// TwinCAT 3 PLC project OPCUA_Client
// Title: OPC UA client
// Company: Hehamala
// Author: Henri Hämäläinen
// ProjectVersion: 0.1
// Description: Tools for utitilizing PLCopen OPCUA functionalities more conveniently
// ProgramVersion: 3.1.4023.0
// libraries:
//   Tc2_Standard, * (Beckhoff Automation GmbH)
//   Tc2_System, * (Beckhoff Automation GmbH)
//   Tc3_Module, * (Beckhoff Automation GmbH)
//   Tc3_PLCopen_OpcUa, * (Beckhoff Automation GmbH)
//   TcUnit, * (www.tcunit.org)
// project tree:
//   / PlcTask.TcTTO
//   POUs/FBs/ FB_OPCUA_ClientConnection.TcPOU, FB_OPCUA_WorkOnNode.TcPOU
//   POUs/FBs/Wrappers/ UA_ConnectWrapper.TcPOU, UA_DisconnectWrapper.TcPOU, UA_GetNameSpaceIndexWrapper.TcPOU, UA_NodeGetHandleWrapper.TcPOU, UA_NodeReleaseHandleWrapper.TcPOU, UA_ReadWrapper.TcPOU, UA_WriteWrapper.TcPOU
//   POUs/ITFs/ I_OPCUA_ClientConnection.TcIO, I_OPCUA_Connect.TcIO, I_OPCUA_Disconnect.TcIO, I_OPCUA_GetNameSpaceIndex.TcIO, I_OPCUA_NodeGetHandle.TcIO, I_OPCUA_NodeReleaseHandle.TcIO, I_OPCUA_Read.TcIO, I_OPCUA_WorkOnNode.TcIO, I_OPCUA_Write.TcIO
//   POUs/Unit tests/ FB_OPCUA_ClientConnection_Test.TcPOU, FB_OPCUA_WorkOnNode_Test.TcPOU, TEST_MAIN.TcPOU
//   POUs/Unit tests/Mocks/ FB_UAconnectMock_Failure.TcPOU, FB_UAconnectMock_Success.TcPOU, FB_UAdisconnectMock_success.TcPOU, FB_UAgetNameSpaceIndexMock_success.TcPOU, FB_UAnodeGetHandleMock_Success.TcPOU, FB_UAnodeReleaseHandleMock_Success.TcPOU, FB_UAreadMock_BoolChangesToTrue.TcPOU, FB_UAwriteMock_Failure.TcPOU
//   Version/ Global_Version.TcGVL
// real-time tasks:
//   TASK PlcTask: cycle T#10ms, priority 20, ADS port 350

CONFIGURATION OPCUA_Client
    RESOURCE PLC ON TwinCAT3
        TASK PlcTask(INTERVAL := T#10ms, PRIORITY := 20);
        PROGRAM TEST_MAIN WITH PlcTask : TEST_MAIN;
    END_RESOURCE
END_CONFIGURATION

// ---- Version/Global_Version.TcGVL
{attribute 'TcGenerated'}
{attribute 'no-analysis'}
{attribute 'linkalways'}
// This function has been automatically generated from the project information.
VAR_GLOBAL CONSTANT
	{attribute 'const_non_replaced'}
	stLibVersion_OPC_UA_client : ST_LibVersion := (iMajor := 0, iMinor := 1, iBuild := 0, iRevision := 0, nFlags := 0, sVersion := '0.1');
END_VAR

// ---- POUs/ITFs/I_OPCUA_ClientConnection.TcIO
INTERFACE I_OPCUA_ClientConnection

METHOD connect : BOOL
VAR_INPUT
	(* server address *)
	serverUrl 		: STRING(MAX_STRING_LENGTH); 
	(* namespace uri*)
	namespaceUri	: STRING(MAX_STRING_LENGTH);
	(* Location of data in namespace *)
	nameSpaceLocationIdentifier : STRING(MAX_STRING_LENGTH);
	(* Session connect info struct *)
	sessionConnectInfo	: ST_UASessionConnectInfo;
END_VAR
END_METHOD

METHOD disconnect : BOOL
END_METHOD

END_INTERFACE

// ---- POUs/ITFs/I_OPCUA_Connect.TcIO
INTERFACE I_OPCUA_Connect

METHOD start : BOOL
VAR_INPUT
    Execute            : BOOL;
    ServerUrl          : STRING(MAX_STRING_LENGTH);
    SessionConnectInfo : ST_UASessionConnectInfo;     
    Timeout            : TIME := DEFAULT_ADS_TIMEOUT; 
END_VAR
VAR_OUTPUT
    ConnectionHdl : DWORD;
    Done          : BOOL;
    Busy          : BOOL;
    Error         : BOOL;
    ErrorID       : DWORD;
END_VAR
END_METHOD

END_INTERFACE

// ---- POUs/ITFs/I_OPCUA_Disconnect.TcIO
INTERFACE I_OPCUA_Disconnect

METHOD start : BOOL
VAR_INPUT
    Execute           : BOOL;
    ConnectionHdl     : DWORD;     
    Timeout           : TIME := DEFAULT_ADS_TIMEOUT; 
END_VAR 
VAR_OUTPUT
    Done        : BOOL;
    Busy        : BOOL;
    Error       : BOOL;
    ErrorID     : DWORD;
END_VAR
END_METHOD

END_INTERFACE

// ---- POUs/ITFs/I_OPCUA_GetNameSpaceIndex.TcIO
INTERFACE I_OPCUA_GetNameSpaceIndex

METHOD start : BOOL
VAR_INPUT
    Execute       : BOOL;
    ConnectionHdl : DWORD;
    NamespaceUri  : STRING(MAX_STRING_LENGTH);
    Timeout       : TIME := DEFAULT_ADS_TIMEOUT; 
END_VAR
VAR_OUTPUT
    NamespaceIndex : UINT;
    Done           : BOOL;
    Busy           : BOOL;
    Error          : BOOL;
    ErrorID        : DWORD;
END_VAR
END_METHOD

END_INTERFACE

// ---- POUs/ITFs/I_OPCUA_NodeGetHandle.TcIO
INTERFACE I_OPCUA_NodeGetHandle

METHOD start : BOOL
VAR_INPUT
    Execute       : BOOL;
    ConnectionHdl : DWORD;
    NodeID        : ST_UANodeID;
    Timeout       : TIME := DEFAULT_ADS_TIMEOUT; 
END_VAR 
VAR_OUTPUT
    NodeHdl     : DWORD;
    Done        : BOOL;
    Busy        : BOOL;
    Error       : BOOL;
    ErrorID     : DWORD;
END_VAR
END_METHOD

END_INTERFACE

// ---- POUs/ITFs/I_OPCUA_NodeReleaseHandle.TcIO
INTERFACE I_OPCUA_NodeReleaseHandle

METHOD start : BOOL
VAR_INPUT
    Execute       : BOOL;
    ConnectionHdl : DWORD;
    NodeHdl       : DWORD;
    Timeout       : TIME := DEFAULT_ADS_TIMEOUT; 
END_VAR 
VAR_OUTPUT
    Done       : BOOL;
    Busy       : BOOL;
    Error      : BOOL;
    ErrorID    : DWORD;
END_VAR
END_METHOD

END_INTERFACE

// ---- POUs/ITFs/I_OPCUA_Read.TcIO
INTERFACE I_OPCUA_Read

METHOD start : BOOL
VAR_INPUT
    Execute           : BOOL;
    ConnectionHdl     : DWORD;
    NodeHdl           : DWORD;
    stNodeAddInfo     : ST_UANodeAdditionalInfo;
    pVariable         : PVOID;
    cbData            : UDINT;
    Timeout           : TIME := DEFAULT_ADS_TIMEOUT;    
END_VAR 
VAR_OUTPUT
    Done        : BOOL;
    Busy        : BOOL;
    Error       : BOOL;
    ErrorID     : UDINT;
    cbData_R    : UDINT;
END_VAR
END_METHOD

END_INTERFACE

// ---- POUs/ITFs/I_OPCUA_WorkOnNode.TcIO
INTERFACE I_OPCUA_WorkOnNode

METHOD read : BOOL
VAR_INPUT
	//clientVariable	: ANY;
	(* VAR_INFO of the target variable (from GVL_OPC)*)
	//clientVariableInfo	: __SYSTEM.VAR_INFO;
	clientVariableAddress	: PVOID;
	clientVariableSize : UDINT;
	serverNodeIdentifier	: STRING;
	nameSpaceLocationIdentifierEx : STRING(MAX_STRING_LENGTH);
	connectionHdl : DWORD;
	nNamespaceIndex			: UINT;
END_VAR
END_METHOD

METHOD write : BOOL
VAR_INPUT
	//clientVariable	: ANY;
	(* VAR_INFO of the target variable (from GVL_OPC)*)
	//clientVariableInfo	: __SYSTEM.VAR_INFO;
	clientVariableAddress	: PVOID;
	clientVariableSize : UDINT;
	serverNodeIdentifier	: STRING;
	nameSpaceLocationIdentifierEx : STRING(MAX_STRING_LENGTH);
	connectionHdl : DWORD;
	nNamespaceIndex			: UINT;
END_VAR
END_METHOD

END_INTERFACE

// ---- POUs/ITFs/I_OPCUA_Write.TcIO
INTERFACE I_OPCUA_Write

METHOD start : BOOL
VAR_INPUT
    Execute        : BOOL;
    ConnectionHdl  : DWORD;
    NodeHdl        : DWORD;
    stNodeAddInfo  : ST_UANodeAdditionalInfo; 
    pVariable      : PVOID;
    cbData         : UDINT;     
    Timeout        : TIME := DEFAULT_ADS_TIMEOUT; 
END_VAR 
VAR_OUTPUT
    Done      : BOOL;
    Busy      : BOOL;
    Error     : BOOL;
    ErrorID   : DWORD;
END_VAR
END_METHOD

END_INTERFACE

// ---- POUs/Unit tests/TEST_MAIN.TcPOU
PROGRAM TEST_MAIN
VAR
	clientConnectionTest 	: FB_OPCUA_ClientConnection_Test;
	workOnNodeTest			: FB_OPCUA_WorkOnNode_Test;
	startTest				: BOOL;
END_VAR


IF startTest THEN
	TcUnit.RUN();
END_IF

END_PROGRAM

// ---- POUs/Unit tests/FB_OPCUA_ClientConnection_Test.TcPOU
FUNCTION_BLOCK FB_OPCUA_ClientConnection_Test  EXTENDS TcUnit.FB_TestSuite
VAR_INPUT
END_VAR
VAR_OUTPUT
END_VAR
VAR
END_VAR

errorShouldntBeActiveWhenConnectionIsSuccesful();
errorShouldBeActiveIfConnectingFails();

METHOD errorShouldBeActiveIfConnectingFails
VAR
	connect 				: FB_UAconnectMock_Failure;
	disconnect 				: FB_UAdisconnectMock_success;
	getNameSpaceIndex 		: FB_UAgetNameSpaceIndexMock_success;
	connection 				: FB_OPCUA_ClientConnection(iOPCUAconnect := connect,
														iOPCUAdisconnect := disconnect,
														iOPCUAgetNameSpaceIndex := getNameSpaceIndex);
	sessionCOnnectInfo 		: ST_UASessionConnectInfo;
END_VAR
TEST('errorShouldBeActiveIfConnectingFails');
	connection.connect(serverUrl := '11.11.11.11',
				namespaceUri := 'namespace',
				nameSpaceLocationIdentifier := 'GVL_ident' ,
				sessionConnectInfo := SessionConnectInfo
				);
	assertEquals_BOOL(Expected := TRUE, Actual := connection.error, Message := 'Error not active when connection failed');
TEST_FINISHED();
END_METHOD

METHOD errorShouldntBeActiveWhenConnectionIsSuccesful
VAR
	connect : FB_UAconnectMock_Success;
	disconnect : FB_UAdisconnectMock_success;
	getNameSpaceIndex : FB_UAgetNameSpaceIndexMock_success;
	connection : FB_OPCUA_ClientConnection(iOPCUAconnect := connect,
										iOPCUAdisconnect := disconnect,
										iOPCUAgetNameSpaceIndex := getNameSpaceIndex);
	sessionCOnnectInfo : ST_UASessionConnectInfo;
END_VAR
TEST('errorShouldntBeActiveWhenConnectionIsSuccesful');
	connection.connect(serverUrl := '11.11.11.11',
				namespaceUri := 'namespace',
				nameSpaceLocationIdentifier := 'GVL_ident' ,
				sessionConnectInfo := SessionConnectInfo
				);
	assertEquals_BOOL(Expected := FALSE, Actual := connection.error, Message := 'Error active even when connection succeeced');
TEST_FINISHED();
END_METHOD

END_FUNCTION_BLOCK

// ---- POUs/Unit tests/Mocks/FB_UAconnectMock_Failure.TcPOU
FUNCTION_BLOCK FB_UAconnectMock_Failure IMPLEMENTS I_OPCUA_Connect
VAR_INPUT
END_VAR
VAR_OUTPUT
END_VAR
VAR
END_VAR

{warning 'add method implementation '}
METHOD start : BOOL
VAR_INPUT
	Execute	: BOOL;
	ServerUrl	: STRING(MAX_STRING_LENGTH);
	SessionConnectInfo	: Tc3_PLCopen_OpcUa.ST_UASessionConnectInfo;
	Timeout	: TIME := DEFAULT_ADS_TIMEOUT;
END_VAR
VAR_OUTPUT
	ConnectionHdl	: DWORD;
	Done	: BOOL;
	Busy	: BOOL;
	Error	: BOOL;
	ErrorID	: DWORD;
END_VAR
IF execute THEN
	error := TRUE;
END_IF
END_METHOD

END_FUNCTION_BLOCK

// ---- POUs/Unit tests/Mocks/FB_UAdisconnectMock_success.TcPOU
FUNCTION_BLOCK FB_UAdisconnectMock_success IMPLEMENTS I_OPCUA_Disconnect
VAR_INPUT
END_VAR
VAR_OUTPUT
END_VAR
VAR
END_VAR

{warning 'add method implementation '}
METHOD start : BOOL
VAR_INPUT
	Execute	: BOOL;
	ConnectionHdl	: DWORD;
	Timeout	: TIME := DEFAULT_ADS_TIMEOUT;
END_VAR
VAR_OUTPUT
	Done	: BOOL;
	Busy	: BOOL;
	Error	: BOOL;
	ErrorID	: DWORD;
END_VAR
IF execute THEN
	done := TRUE;
END_IF
END_METHOD

END_FUNCTION_BLOCK

// ---- POUs/Unit tests/Mocks/FB_UAgetNameSpaceIndexMock_success.TcPOU
FUNCTION_BLOCK FB_UAgetNameSpaceIndexMock_success IMPLEMENTS I_OPCUA_GetNameSpaceIndex
VAR_INPUT
END_VAR
VAR_OUTPUT
END_VAR
VAR
END_VAR

{warning 'add method implementation '}
METHOD start : BOOL
VAR_INPUT
	Execute	: BOOL;
	ConnectionHdl	: DWORD;
	NamespaceUri	: STRING(MAX_STRING_LENGTH);
	Timeout	: TIME := DEFAULT_ADS_TIMEOUT;
END_VAR
VAR_OUTPUT
	NamespaceIndex	: UINT;
	Done	: BOOL;
	Busy	: BOOL;
	Error	: BOOL;
	ErrorID	: DWORD;
END_VAR
IF execute THEN
	done := TRUE;
END_IF
END_METHOD

END_FUNCTION_BLOCK

// ---- POUs/FBs/FB_OPCUA_ClientConnection.TcPOU
FUNCTION_BLOCK FB_OPCUA_ClientConnection IMPLEMENTS I_OPCUA_ClientConnection
VAR_INPUT
END_VAR
VAR_OUTPUT
	connectionHdl : DWORD;
	nNamespaceIndex			: UINT;
	connectDone : BOOL;
	disconnectDone : BOOL;
	error : BOOL;
END_VAR
VAR
	nameSpaceLocationIdentifierEx : STRING(MAX_STRING_LENGTH); 
	NamespaceUriEx : STRING(MAX_STRING_LENGTH); 
	
	{IF defined (Test)}	
		_iOPCUA_Connect				: I_OPCUA_COnnect;
		_iOPCUA_GetNameSpaceIndex 	: I_OPCUA_GetNameSpaceIndex;
		_iOPCUA_Disconnect			: I_OPCUA_Disconnect;
	{ELSE}
		_iOPCUA_Connect				: UA_ConnectWrapper;		
		_iOPCUA_GetNameSpaceIndex 	: UA_GetNameSpaceIndexWrapper;
		_iOPCUA_Disconnect			: UA_DisconnectWrapper;
	{END_IF}
		
	SessionConnectInfoEx	: ST_UASessionConnectInfo;
	
	

	
	(* Other declarations *) 
	errorID : DWORD;	
	executing : BOOL;
	firstTimeWrite : BOOL;
	serverURLex: STRING(MAX_STRING_LENGTH);
	connectStep: INT;
	disconnectStep: INT;
	connectBusy: BOOL;
	connectError: BOOL;
	getNameSpaceIndexBusy: BOOL;
	getNameSpaceIndexError: BOOL;
	disconnectBusy: BOOL;
	disconnectError: BOOL;
	getNameSpaceErrorID: DWORD;
	connectErrorID: DWORD;
END_VAR

{warning 'add method implementation '}
METHOD connect : BOOL
VAR_INPUT
	(* server address *)
	serverUrl	: STRING(MAX_STRING_LENGTH);
	(* namespace uri*)
	namespaceUri	: STRING(MAX_STRING_LENGTH);
	(* Location of data in namespace *)
	nameSpaceLocationIdentifier	: STRING(MAX_STRING_LENGTH);
	(* Session connect info struct *)
	sessionConnectInfo	: ST_UASessionConnectInfo;
END_VAR


CASE connectStep OF
	0:
		error := FALSE;
		connectDone := FALSE;
		disconnectStep := 0;
		nameSpaceUriEx := namespaceUri;
		sessionConnectInfoEx := SessionConnectInfo;
		serverURlex := serverUrl;
		nameSpaceLocationIdentifierEx := nameSpaceLocationIdentifier;
		SessionConnectInfoEx.sApplicationName := 'asddddd';
		_iOPCUA_Connect.start(
			Execute				:= TRUE,
			ServerURL			:= serverURLex,
			SessionConnectInfo  := SessionConnectInfoEx,
			Timeout				:= T#2M,
			ConnectionHdl		=> ConnectionHdl,
			busy				=> connectBusy,
			error				=> connectError,
			errorID				=> connectErrorID
		);
		IF NOT connectBusy THEN
			_iOPCUA_Connect.start(Execute := FALSE,
								ServerURL			:= serverURLex,
								SessionConnectInfo  := SessionConnectInfoEx,
								Timeout				:= T#2M,
								ConnectionHdl		=> ConnectionHdl
								);
	
			IF NOT connectError THEN
				(* session open *)
				connectStep :=connectStep + 1;
			ELSE
				Error			:= TRUE;
				ErrorID		:= connectErrorID;
				ConnectionHdl	:= 0;
				connectStep		:= 0; (* idle *)
			END_IF
		END_IF
	1:
		_iOPCUA_GetNameSpaceIndex.start(
										Execute			:= TRUE,
										ConnectionHdl	:= ConnectionHdl,
										NamespaceUri	:= NamespaceUriEx,
										TimeOut 		:= T#5S,
										NamespaceIndex	=> nNamespaceIndex,
										busy			=> getNameSpaceIndexBusy,
										error			=> getNameSpaceIndexError,
										errorID			=> getNameSpaceErrorID
										);
	
	
		IF NOT getNameSpaceIndexBusy THEN
			_iOPCUA_GetNameSpaceIndex.start(Execute := FALSE,
											ConnectionHdl	:= ConnectionHdl,
											NamespaceUri	:= NamespaceUriEx,
											TimeOut 		:= T#5S,
											NamespaceIndex	=> nNamespaceIndex,
											);
			IF NOT getNameSpaceIndexError THEN
				(* session closed *)
				connectDone := TRUE;
				connectStep 	:= 0; (* idle *)
			ELSE
				Error		:= TRUE;
				ErrorID	:= getNameSpaceErrorID;
				connectStep := 0;
				// CLEANUP?writeStep 		:= 5; (* idle *)
			END_IF
		END_IF	
END_CASE
END_METHOD

{warning 'add method implementation '}
METHOD disconnect : BOOL

VAR
	Execute: INT;
	disconnectErrorID: DWORD;
END_VAR
CASE disconnectStep OF
	0:	(* close session *)
		error := FALSE;
		disconnectDone := FALSE;
		connectStep := 0;
		_iOPCUA_Disconnect.start(
							Execute			:= TRUE,
							ConnectionHdl	:= connectionHdl,
							timeOut			:= T#5S,
							busy			=> disconnectBusy,
							error			=> disconnectError,
							errorID			=> disconnectErrorID
						);
	
		IF NOT disconnectBusy THEN
			_iOPCUA_Disconnect.start(Execute := FALSE,
									ConnectionHdl	:= connectionHdl,
									timeOut			:= T#5S
									);
			//Busy := FALSE;
			IF NOT disconnectError THEN
				(* session closed *)
				firstTimeWrite := TRUE;
				Executing := FALSE;
				ConnectionHdl	:= 0; //ADDED
				disconnectStep 		:= 0; (* idle *)
				IF NOT error THEN 
					disconnectDone := TRUE;
					disconnectStep := 0;
				END_IF
			ELSE
				error			:= TRUE;
				errorID		:= disconnectErrorID;
				connectionHdl	:= 0;
				disconnectStep 		:= 0; 
			END_IF
		END_IF	
END_CASE
END_METHOD

METHOD FB_init : BOOL
VAR_INPUT
	bInitRetains					: BOOL; // if TRUE, the retain variables are initialized (warm start / cold start)
	bInCopyCode 					: BOOL;  // if TRUE, the instance afterwards gets moved into the copy code (online change)
	{IF defined (Test)}
		iOPCUAconnect 					: I_OPCUA_Connect;
		iOPCUAdisconnect 				: I_OPCUA_Disconnect;
		iOPCUAgetNameSpaceIndex 		: I_OPCUA_GetNameSpaceIndex; 
	{ END_IF }
END_VAR
{IF defined (Test)}
	_iOPCUA_Connect := iOPCUAconnect;
	_iOPCUA_Disconnect := iOPCUAdisconnect;
	_iOPCUA_GetNameSpaceIndex := iOPCUAgetNameSpaceIndex;
{ END_IF }
END_METHOD

END_FUNCTION_BLOCK

// ---- POUs/FBs/Wrappers/UA_ConnectWrapper.TcPOU
FUNCTION_BLOCK UA_ConnectWrapper IMPLEMENTS I_OPCUA_Connect
VAR_INPUT
END_VAR
VAR_OUTPUT
END_VAR
VAR
	uaConnect : UA_Connect;
END_VAR

{warning 'add method implementation '}
METHOD start : BOOL
VAR_INPUT
	Execute					: BOOL;
	ServerUrl				: STRING(MAX_STRING_LENGTH);
	SessionConnectInfo		: Tc3_PLCopen_OpcUa.ST_UASessionConnectInfo;
	Timeout					: TIME := DEFAULT_ADS_TIMEOUT;
END_VAR
VAR_OUTPUT
	ConnectionHdl			: DWORD;
	Done					: BOOL;
	Busy					: BOOL;
	Error					: BOOL;
	ErrorID					: DWORD;
END_VAR
uaConnect(Execute					:= Execute,
          ServerUrl				:= ServerUrl	,
          SessionConnectInfo		:= SessionConnectInfo,
          Timeout					:= Timeout,
		  ConnectionHdl			=> ConnectionHdl,
		  Done					=> Done,
          Busy					=> Busy,
          Error					=> Error,
          ErrorID				=> ErrorID
		  );
END_METHOD

END_FUNCTION_BLOCK

// ---- POUs/FBs/Wrappers/UA_GetNameSpaceIndexWrapper.TcPOU
FUNCTION_BLOCK UA_GetNameSpaceIndexWrapper IMPLEMENTS I_OPCUA_GetNameSpaceIndex
VAR_INPUT
END_VAR
VAR_OUTPUT
END_VAR
VAR
	uaGetNameSpaceIndex : UA_GetNameSpaceIndex;
END_VAR

{warning 'add method implementation '}
METHOD start : BOOL
VAR_INPUT
	Execute			: BOOL;
	ConnectionHdl	: DWORD;
	NamespaceUri	: STRING(MAX_STRING_LENGTH);
	Timeout			: TIME := DEFAULT_ADS_TIMEOUT;
END_VAR
VAR_OUTPUT
	NamespaceIndex	: UINT;
	Done			: BOOL;
	Busy			: BOOL;
	Error			: BOOL;
	ErrorID			: DWORD;
END_VAR
uaGetNameSpaceIndex(Execute			:= Execute,
                    ConnectionHdl	:= ConnectionHdl,
                    NamespaceUri	:= Namespaceuri,
                    Timeout			:= Timeout,
					NamespaceIndex	=> NamespaceIndex,
                    Done			=> Done,
                    Busy			=> Busy,
                    Error			=> Error,
                    ErrorID			=> ErrorID);
END_METHOD

END_FUNCTION_BLOCK

// ---- POUs/FBs/Wrappers/UA_DisconnectWrapper.TcPOU
FUNCTION_BLOCK UA_DisconnectWrapper IMPLEMENTS I_OPCUA_Disconnect
VAR_INPUT
END_VAR
VAR_OUTPUT
END_VAR
VAR
	uaDisconnect : UA_Disconnect;
END_VAR

{warning 'add method implementation '}
METHOD start : BOOL
VAR_INPUT
	Execute			: BOOL;
	ConnectionHdl	: DWORD;
	Timeout			: TIME := DEFAULT_ADS_TIMEOUT;
END_VAR
VAR_OUTPUT
	Done	: BOOL;
	Busy	: BOOL;
	Error	: BOOL;
	ErrorID	: DWORD;
END_VAR
uaDisconnect(Execute			:= Execute,
             ConnectionHdl	:= ConnectionHdl,
             Timeout			:= Timeout,
			 Done			=> Done,
			 Busy			=> Busy,
             Error			=> Error,
             ErrorID 		=> ErrorID);
END_METHOD

END_FUNCTION_BLOCK

// ---- POUs/Unit tests/Mocks/FB_UAconnectMock_Success.TcPOU
FUNCTION_BLOCK FB_UAconnectMock_Success IMPLEMENTS I_OPCUA_Connect
VAR_INPUT
END_VAR
VAR_OUTPUT
END_VAR
VAR
END_VAR

{warning 'add method implementation '}
METHOD start : BOOL
VAR_INPUT
	Execute	: BOOL;
	ServerUrl	: STRING(MAX_STRING_LENGTH);
	SessionConnectInfo	: Tc3_PLCopen_OpcUa.ST_UASessionConnectInfo;
	Timeout	: TIME := DEFAULT_ADS_TIMEOUT;
END_VAR
VAR_OUTPUT
	ConnectionHdl	: DWORD;
	Done	: BOOL;
	Busy	: BOOL;
	Error	: BOOL;
	ErrorID	: DWORD;
END_VAR
IF execute THEN
	done := TRUE;
END_IF
END_METHOD

END_FUNCTION_BLOCK

// ---- POUs/Unit tests/FB_OPCUA_WorkOnNode_Test.TcPOU
FUNCTION_BLOCK FB_OPCUA_WorkOnNode_Test  EXTENDS TcUnit.FB_TestSuite
VAR_INPUT
END_VAR
VAR_OUTPUT
END_VAR
VAR
	read	 				: FB_UAreadMock_BoolChangesToTrue;
	write					: FB_UAwriteMock_Failure;
	nodeReleaseHandle		: FB_UAnodeReleaseHandleMock_Success;
	nodeGetHandle			: FB_UAnodeGetHandleMock_Success;

	readNode 				: FB_OPCUA_WorkOnNode(
													iOPCUA_Write := write,			
													iOPCUA_Read	:= read,				
													iOPCUA_NodeReleaseHandle := nodeReleaseHandle,	
													iOPCUA_NodeGetHandle :=  nodeGetHandle		
													);
	booleanToRead : BOOL;
	booleanInfo : __SYSTEM.VAR_INFO := __VARINFO(readNode);
END_VAR

variableShouldGetUpdatedWhenChanged();

METHOD errorShouldActivateIfWriteFails
VAR
	sessionCOnnectInfo 		: ST_UASessionConnectInfo;
END_VAR
END_METHOD

METHOD variableShouldGetUpdatedWhenChanged
VAR
	sessionCOnnectInfo 		: ST_UASessionConnectInfo;
END_VAR
TEST('variableShouldGetUpdatedWhenChanged');
	
	
	readNode.read(//clientVariable := booleanToRead,
					clientVariableAddress := ADR(booleanToRead),
					clientVariableSize := SIZEOF(booleanToRead),
					serverNodeIdentifier := 'test',
					nameSpaceLocationIdentifierEx := 'test',
					ConnectionHdl := 11,
					nNamespaceIndex := 11);
	IF NOT readNode.busy THEN
		assertEquals_BOOL(Expected := TRUE, Actual := booleanToRead, Message := 'Value not updated when changed');
		TEST_FINISHED();
	END_IF
END_METHOD

END_FUNCTION_BLOCK

// ---- POUs/Unit tests/Mocks/FB_UAreadMock_BoolChangesToTrue.TcPOU
FUNCTION_BLOCK FB_UAreadMock_BoolChangesToTrue IMPLEMENTS I_OPCUA_Read
VAR_INPUT
END_VAR
VAR_OUTPUT
END_VAR
VAR
END_VAR

{warning 'add method implementation '}
METHOD start : BOOL
VAR_INPUT
	Execute	: BOOL;
	ConnectionHdl	: DWORD;
	NodeHdl	: DWORD;
	stNodeAddInfo	: Tc3_PLCopen_OpcUa.ST_UANodeAdditionalInfo;
	pVariable	: PVOID;
	cbData	: UDINT;
	Timeout	: TIME := DEFAULT_ADS_TIMEOUT;
END_VAR
VAR_OUTPUT
	Done	: BOOL;
	Busy	: BOOL;
	Error	: BOOL;
	ErrorID	: UDINT;
	cbData_R	: UDINT;
END_VAR
IF execute THEN
	MEMSET(pVariable,1,SIZEOF(cbData));
	done := TRUE;
END_IF
END_METHOD

END_FUNCTION_BLOCK

// ---- POUs/Unit tests/Mocks/FB_UAwriteMock_Failure.TcPOU
FUNCTION_BLOCK FB_UAwriteMock_Failure IMPLEMENTS I_OPCUA_Write
VAR_INPUT
END_VAR
VAR_OUTPUT
END_VAR
VAR
END_VAR

{warning 'add method implementation '}
METHOD start : BOOL
VAR_INPUT
	Execute	: BOOL;
	ConnectionHdl	: DWORD;
	NodeHdl	: DWORD;
	stNodeAddInfo	: Tc3_PLCopen_OpcUa.ST_UANodeAdditionalInfo;
	pVariable	: PVOID;
	cbData	: UDINT;
	Timeout	: TIME := DEFAULT_ADS_TIMEOUT;
END_VAR
VAR_OUTPUT
	Done	: BOOL;
	Busy	: BOOL;
	Error	: BOOL;
	ErrorID	: DWORD;
END_VAR
IF execute THEN
	Error := TRUE;
END_IF
END_METHOD

END_FUNCTION_BLOCK

// ---- POUs/Unit tests/Mocks/FB_UAnodeReleaseHandleMock_Success.TcPOU
FUNCTION_BLOCK FB_UAnodeReleaseHandleMock_Success IMPLEMENTS I_OPCUA_NodeReleaseHandle
VAR_INPUT
END_VAR
VAR_OUTPUT
END_VAR
VAR
END_VAR

{warning 'add method implementation '}
METHOD start : BOOL
VAR_INPUT
    Execute       : BOOL;
    ConnectionHdl : DWORD;
    NodeHdl       : DWORD;
    Timeout       : TIME := DEFAULT_ADS_TIMEOUT; 
END_VAR
VAR_OUTPUT
	Done	: BOOL;
	Busy	: BOOL;
	Error	: BOOL;
	ErrorID	: DWORD;
END_VAR
IF execute THEN
	done := TRUE;
END_IF
END_METHOD

END_FUNCTION_BLOCK

// ---- POUs/Unit tests/Mocks/FB_UAnodeGetHandleMock_Success.TcPOU
FUNCTION_BLOCK FB_UAnodeGetHandleMock_Success IMPLEMENTS I_OPCUA_NodeGetHandle
VAR_INPUT
END_VAR
VAR_OUTPUT
END_VAR
VAR
END_VAR

{warning 'add method implementation '}
METHOD start : BOOL
VAR_INPUT
	Execute	: BOOL;
	ConnectionHdl	: DWORD;
	NodeID	: Tc3_PLCopen_OpcUa.ST_UANodeID;
	Timeout	: TIME := DEFAULT_ADS_TIMEOUT;
END_VAR
VAR_OUTPUT
	NodeHdl	: DWORD;
	Done	: BOOL;
	Busy	: BOOL;
	Error	: BOOL;
	ErrorID	: DWORD;
END_VAR
IF execute THEN
	Done := TRUE;
END_IF
END_METHOD

END_FUNCTION_BLOCK

// ---- POUs/FBs/FB_OPCUA_WorkOnNode.TcPOU
FUNCTION_BLOCK FB_OPCUA_WorkOnNode IMPLEMENTS I_OPCUA_WorkOnNode
VAR_INPUT
END_VAR
VAR_OUTPUT
	busy: BOOL;
	error : BOOL;
END_VAR
VAR

	stNodeAddInfo			: ST_UANodeAdditionalInfo;
	cbData_R				: UDINT;
	
	iState		: INT;
	nErrorID	: DWORD;
	lastErrorStep: INT;
	Executing : BOOL;
	writeStep : INT;
	(* Declarations for UA_Write *)
	{IF defined (Test)}
		_iOPCUA_Write : I_OPCUA_Write; 
		(* Declarations for UA_NodeReleaseHandle *)
		_iOPCUA_NodeReleaseHandle : I_OPCUA_NodeReleaseHandle;
		_iOPCUA_NodeGetHandle : I_OPCUA_NodeGetHandle;
		_iOPCUA_Read			: I_OPCUA_Read;
	{ELSE}
		_iOPCUA_Write : UA_WriteWrapper;
		_iOPCUA_NodeReleaseHandle : UA_NOdeReleaseHandleWrapper;
		_iOPCUA_NodeGetHandle : UA_NodeGetHandleWrapper;
		_iOPCUA_Read			: UA_ReadWrapper;
	{ END_IF}
	(* Other declarations *) 
	errorID : DWORD;	
	clientVariablePrev : BYTE;
	firstTimeWrite : BOOL;
	//_iOPCUA_NodeGetHandle : I_OPCUA_NodeGetHandle;
	NodeID : ST_UANodeID;
	nNodeHdl : DWORD;
	NodeGetHandleBusy: BOOL;
	NodeGetHandleError: BOOL;
	NodeGetHandleErrorID: DWORD;
	readBusy: BOOL;
	readError: BOOL;
	readErrorID: DWORD;
	nodeReleaseHandleBusy: BOOL;
	nodeReleaseHandleError: BOOL;
	nodeReleaseHandleErrorID: DWORD;
	writeBusy: BOOL;
	writeError: BOOL;
	writeErrorID: DWORD;
	clientVarInfo : __SYSTEM.VAR_INFO;
	pClientByteValue : POINTER TO BYTE;
	ConnectionHdlPrev: DWORD;
END_VAR

METHOD FB_init : BOOL
VAR_INPUT
	bInitRetains : BOOL; // if TRUE, the retain variables are initialized (warm start / cold start)
	bInCopyCode : BOOL;  // if TRUE, the instance afterwards gets moved into the copy code (online change)
	{IF defined (Test)}
		iOPCUA_Write				: I_OPCUA_Write;
		iOPCUA_Read					: I_OPCUA_Read;
		iOPCUA_NodeReleaseHandle 	: I_OPCUA_NodeReleaseHandle;
		iOPCUA_NodeGetHandle 		: I_OPCUA_NodeGetHandle;
	{END_IF}
END_VAR
{IF defined (Test)}
	_iOPCUA_Write	:= iOPCUA_Write;		
	_iOPCUA_Read		:= iOPCUA_Read	;		
	_iOPCUA_NodeReleaseHandle := iOPCUA_NodeReleaseHandle;
	_iOPCUA_NodeGetHandle 	:= iOPCUA_NodeGetHandle 	;
{END_IF}
END_METHOD

{warning 'add method implementation '}
METHOD read : BOOL
VAR_INPUT
	{attribute 'anytypeclass' := 'ANY'}
	//clientVariable	: ANY;
	(* VAR_INFO of the target variable (from GVL_OPC)*)
	//clientVariableInfo	: __SYSTEM.VAR_INFO;
	clientVariableAddress : PVOID;
	clientVariableSize : UDINT;
	serverNodeIdentifier	: STRING;
	nameSpaceLocationIdentifierEx	: STRING(MAX_STRING_LENGTH);
	ConnectionHdl	: DWORD;
	nNamespaceIndex			: UINT;
END_VAR

IF ConnectionHdl <> ConnectionHdlPrev THEN
	istate := 0;
	ConnectionHdlPrev := ConnectionHdl;
	error := FALSE;
END_IF

CASE istate OF
0: 
		error := FALSE;
		nNodeHdl :=0;
		iState := iState + 1;
		Executing := TRUE;
	
1:	(* Get Node Handle *)
	
		NodeID.eIdentifierType := eUAIdentifierType_String;
		NodeID.nNamespaceIndex := nNamespaceIndex;
		NodeID.sIdentifier := CONCAT(nameSpaceLocationIdentifierEx,serverNodeIdentifier);
		_iOPCUA_NodeGetHandle.start(
									Execute := TRUE,
									ConnectionHdl := connectionHdl,
									NodeID := NodeID,
									Timeout := T#5S,
									NodeHdl => nNodeHdl,
									Busy => NodeGetHandleBusy,
									Error => NodeGetHandleError,
									ErrorID => NodeGetHandleErrorID
									);
		IF NOT NodeGetHandleBusy THEN
		  _iOPCUA_NodeGetHandle.start(Execute := FALSE,
										ConnectionHdl := connectionHdl,
										NodeID := NodeID,
										Timeout := T#5S
										);
		  IF NOT NodeGetHandleError THEN
			istate := istate + 1;
		  ELSE
			errorID := NodeGetHandleErrorID;
			istate := 3;
		  END_IF
		END_IF

	
2: 	(* UA_Read *)

	//dataAdd := ADR(clientVariable);
	clientVarInfo := __VARINFO(clientVariableAddress);
	_iOPCUA_Read.start(
						Execute := TRUE,
						ConnectionHdl := connectionHdl,
						NodeHdl := nNodeHdl,
						cbData := clientVariableSize,//clientVarInfo.BitSize,//SIZEOF(clientVariable),//clientVariableInfo.BitSize,
						stNodeAddInfo 	:= stNodeAddInfo,
						pVariable := clientVariableAddress,//clientVariableInfo.ByteAddress,
						Timeout := T#5S,
						busy => readBusy,
						error => readError,
						errorID => readErrorID,
						cbData_R => cbData_R
						);

	IF NOT readBusy THEN
			_iOPCUA_Read.start( Execute := FALSE, 
						ConnectionHdl := connectionHdl,
						NodeHdl := nNodeHdl,
						cbData := clientVarInfo.BitSize,//SIZEOF(clientVariable),//clientVariableInfo.BitSize,
						stNodeAddInfo 	:= stNodeAddInfo,
						pVariable :=clientVariableAddress,//clientVariableInfo.ByteAddress,
						Timeout := T#5S,
						cbData_R => cbData_R);

		IF NOT readError THEN
			iState 		:= 3;
		ELSE
			lastErrorStep := 2;
			nErrorID	:= readErrorId;
			iState 		:= 3; (* idle *)
		END_IF
	END_IF


3:	(* Release Node Handle *)
		_iOPCUA_NodeReleaseHandle.start(
			Execute			:= TRUE,
			ConnectionHdl	:= ConnectionHdl,
			NodeHdl			:= nNodeHdl,
			Timeout := T#5S,
			busy => nodeReleaseHandleBusy,
			error => nodeReleaseHandleError,
			errorID => nodeReleaseHandleErrorID
		);
	
		IF NOT nodeReleaseHandleBusy THEN
			_iOPCUA_NodeReleaseHandle.start(Execute := FALSE,
											ConnectionHdl	:= ConnectionHdl,
											NodeHdl			:= nNodeHdl,
											Timeout := T#5S
											);
	
			IF NOT nodeReleaseHandleError THEN
				Executing := FALSE;
				istate := 0;
			ELSE
				error := TRUE;
				errorID	:= nodeReleaseHandleErrorID;
				istate 	:= 0; (* idle *)
			END_IF
		END_IF
END_CASE
busy := Executing;
END_METHOD

{warning 'add method implementation '}
METHOD write : BOOL
VAR_INPUT
	{attribute 'anytypeclass' := 'ANY'}
	//clientVariable	: ANY;
	(* VAR_INFO of the target variable (from GVL_OPC)*)
	//clientVariableInfo	: __SYSTEM.VAR_INFO;
	clientVariableAddress	: PVOID;
	clientVariableSize : UDINT;
	serverNodeIdentifier	: STRING;
	nameSpaceLocationIdentifierEx	: STRING(MAX_STRING_LENGTH);
	connectionHdl: DWORD;
	nNamespaceIndex			: UINT;
END_VAR

IF ConnectionHdl <> ConnectionHdlPrev THEN
	writeStep := 0;
	ConnectionHdlPrev := ConnectionHdl;
	error := FALSE;
	firstTimeWrite := FALSE;
END_IF

CASE writeStep OF
	
	0:
		error := FALSE;
		clientVarInfo := __VARINFO(clientVariableAddress);
		pClientByteValue := clientVariableAddress;
		nNodeHdl := 0;
		//MEMSET(ADR(clientByteValue), clientVarInfo.ByteAddress ,clientVarInfo.BitSize);
		//IF clientVariable.pValue^ <> clientVariablePrev OR NOT firstTimeWrite THEN
		IF pClientByteValue^ <> clientVariablePrev OR NOT firstTimeWrite THEN
			Executing := TRUE;
			clientVariablePrev := pClientByteValue^;
			writeStep := 1;
		END_IF
	
	  1: 
		(* UA_NodeGetHandle *)
		NodeID.eIdentifierType := eUAIdentifierType_String;
		NodeID.nNamespaceIndex := nNamespaceIndex;
		NodeID.sIdentifier := CONCAT(nameSpaceLocationIdentifierEx,serverNodeIdentifier);
		_iOPCUA_NodeGetHandle.start(
									Execute := TRUE,
									ConnectionHdl := connectionHdl,
									NodeID := NodeID,
									Timeout := T#5S,
									NodeHdl => nNodeHdl,
									Busy => nodeGetHandleBusy,
									Error => nodeGetHandleError,
									ErrorID => nodeGetHandleErrorID
									
									);
		IF NOT nodeGetHandleBusy THEN
		  _iOPCUA_NodeGetHandle.start(Execute := FALSE,
									ConnectionHdl := connectionHdl,
									NodeID := NodeID,
									Timeout := T#5S,);
		  IF NOT nodeGetHandleError THEN
			writeStep := writeStep + 1;
		  ELSE
			errorID := nodeGetHandleErrorID;
			writeStep := 2;
		  END_IF
		END_IF
	  2: (* UA_Write *)
		_iOPCUA_Write.start(
							Execute := TRUE,
							ConnectionHdl := connectionHdl,
							NodeHdl := nNodeHdl,
							stNodeAddInfo := stNodeAddInfo,
							cbData := clientVariableSize,//clientVarInfo.BitSize,//SIZEOF(clientVariable),//clientVariableInfo.BitSize,
							pVariable := clientVariableAddress,//clientVariableInfo.ByteAddress,
							Timeout := T#5S,
							busy => writeBusy,
							error => writeError,
							errorID => writeErrorID
							);
		IF NOT writeBusy THEN
		  _iOPCUA_Write.start(
								Execute := FALSE,
								ConnectionHdl := connectionHdl,
								NodeHdl := nNodeHdl,
								stNodeAddInfo := stNodeAddInfo,
								cbData := clientVarInfo.BitSize,//SIZEOF(clientVariable), //clientVariableInfo.BitSize,
								pVariable := clientVariableAddress,//clientVariableInfo.ByteAddress,
								Timeout := T#5S );

		  IF NOT writeError THEN
				writeStep := 3;
		  ELSE
			//Executing := FALSE;
			//error := TRUE;
			errorID := writeErrorID;
			writeStep := 3;
		  END_IF
		END_IF
	3:	(* Release Node Handle *)
		_iOPCUA_NodeReleaseHandle.start(
			Execute			:= TRUE,
			ConnectionHdl	:= ConnectionHdl,
			NodeHdl			:= nNodeHdl,
			TimeOut			:= T#5S,
			Busy			=> nodeReleaseHandleBusy,
			Error			=> nodeReleaseHandleError,
			ErrorID			=> nodeReleaseHandleErrorID
		);
	
		IF NOT nodeReleaseHandleBusy THEN
			_iOPCUA_NodeReleaseHandle.start(Execute := FALSE,
											ConnectionHdl	:= ConnectionHdl,
											NodeHdl			:= nNodeHdl,
											TimeOut			:= T#5S
												);
	
			IF NOT nodeReleaseHandleError THEN
				firstTimeWrite := TRUE;
				Executing := FALSE;
				writeStep := 0;
			ELSE
				error := TRUE;
				errorID	:= nodeReleaseHandleErrorID;
				writeStep 	:= 0; (* idle *)
			END_IF
		END_IF
END_CASE
busy := Executing ;
END_METHOD

END_FUNCTION_BLOCK

// ---- POUs/FBs/Wrappers/UA_WriteWrapper.TcPOU
FUNCTION_BLOCK UA_WriteWrapper IMPLEMENTS I_OPCUA_Write
VAR_INPUT
END_VAR
VAR_OUTPUT
END_VAR
VAR
	uaWrite : UA_Write;
END_VAR

{warning 'add method implementation '}
METHOD start : BOOL
VAR_INPUT
	Execute	: BOOL;
	ConnectionHdl	: DWORD;
	NodeHdl	: DWORD;
	stNodeAddInfo	: Tc3_PLCopen_OpcUa.ST_UANodeAdditionalInfo;
	pVariable	: PVOID;
	cbData	: UDINT;
	Timeout	: TIME := DEFAULT_ADS_TIMEOUT;
END_VAR
VAR_OUTPUT
	Done	: BOOL;
	Busy	: BOOL;
	Error	: BOOL;
	ErrorID	: DWORD;
END_VAR
uaWrite(Execute := execute,
		 COnnectionhdl := connectionhdl, 
		NodeHdl := nodehdl, 
		stNodeAddInfo := stnodeaddinfo, 
		pVariable := pvariable, 
		cbdata := cbData, 
		Timeout := timeout,
		Done => DOne,
		Busy => Busy,
		Error => Error,
		ErrorID => ErrorID
		);
END_METHOD

END_FUNCTION_BLOCK

// ---- POUs/FBs/Wrappers/UA_NodeReleaseHandleWrapper.TcPOU
FUNCTION_BLOCK UA_NodeReleaseHandleWrapper IMPLEMENTS I_OPCUA_NodeReleaseHandle
VAR_INPUT
END_VAR
VAR_OUTPUT
END_VAR
VAR
	uaNodeReleaseHandle : UA_NodeReleaseHandle;
END_VAR

{warning 'add method implementation '}
METHOD start : BOOL
VAR_INPUT
	Execute	: BOOL;
	ConnectionHdl	: DWORD;
	NodeHdl	: DWORD;
	Timeout	: TIME := DEFAULT_ADS_TIMEOUT;
END_VAR
VAR_OUTPUT
	Done	: BOOL;
	Busy	: BOOL;
	Error	: BOOL;
	ErrorID	: DWORD;
END_VAR
uaNodeReleasehandle(Execute := execute, 
					connectionhdl := connectionhdl, 
					nodehdl := nodehdl, 
					timeout := timeout,
					Done => Done,
					Busy => Busy,
					Error => Error,
					ErrorID => ErrorID);
END_METHOD

END_FUNCTION_BLOCK

// ---- POUs/FBs/Wrappers/UA_NodeGetHandleWrapper.TcPOU
FUNCTION_BLOCK UA_NodeGetHandleWrapper IMPLEMENTS I_OPCUA_NodeGetHandle
VAR_INPUT
END_VAR
VAR_OUTPUT
END_VAR
VAR
	uaNodegethandle : UA_NodeGetHandle;
END_VAR

{warning 'add method implementation '}
METHOD start : BOOL
VAR_INPUT
	Execute	: BOOL;
	ConnectionHdl	: DWORD;
	NodeID	: Tc3_PLCopen_OpcUa.ST_UANodeID;
	Timeout	: TIME := DEFAULT_ADS_TIMEOUT;
END_VAR
VAR_OUTPUT
	NodeHdl	: DWORD;
	Done	: BOOL;
	Busy	: BOOL;
	Error	: BOOL;
	ErrorID	: DWORD;
END_VAR
uaNodegethandle(Execute := execute, 
				connectionhdl := connectionhdl, 
				nodeid := nodeid, 
				timeout := timeout,
				NodeHdl => NodeHdl,
				Done => Done,
				Busy => Busy,
				Error => Error,
				ErrorID => ErrorId);
END_METHOD

END_FUNCTION_BLOCK

// ---- POUs/FBs/Wrappers/UA_ReadWrapper.TcPOU
FUNCTION_BLOCK UA_ReadWrapper IMPLEMENTS I_OPCUA_Read
VAR_INPUT
END_VAR
VAR_OUTPUT
END_VAR
VAR
	uaRead : UA_Read;
END_VAR

{warning 'add method implementation '}
METHOD start : BOOL
VAR_INPUT
	Execute	: BOOL;
	ConnectionHdl	: DWORD;
	NodeHdl	: DWORD;
	stNodeAddInfo	: Tc3_PLCopen_OpcUa.ST_UANodeAdditionalInfo;
	pVariable	: PVOID;
	cbData	: UDINT;
	Timeout	: TIME := DEFAULT_ADS_TIMEOUT;
END_VAR
VAR_OUTPUT
	Done	: BOOL;
	Busy	: BOOL;
	Error	: BOOL;
	ErrorID	: UDINT;
	cbData_R	: UDINT;
END_VAR
uaread(Execute := execute,
		 COnnectionhdl := connectionhdl, 
		NodeHdl := nodehdl, 
		stNodeAddInfo := stnodeaddinfo, 
		pVariable := pvariable, 
		cbdata := cbData, 
		Timeout := timeout,
		Done => DOne,
		Busy => Busy,
		Error => Error,
		ErrorID => ErrorID,
		cbData_R => cbData_R
		);
END_METHOD

END_FUNCTION_BLOCK
